TYPE ST_SequenceOut :
STRUCT
END_STRUCT
END_TYPE

(* stored: Version 1.1.0.1
   DUT ST_SequenceOut: Id {4274038c-a6b5-0b31-32b3-4831a7f3fe80} *)
